//=============================================================================
// ST10_Flow4_B1Press.scl
// 1:1 CONVERSION FROM TIA PORTAL V18 GRAPH XML
// Generated: 2026-02-02
//=============================================================================

TYPE
    E_STEP_ST10_Flow4_B1Press : (
        STEP_ST10_Flow4_B1Press_F4_Initial := 1,
        STEP_ST10_Flow4_B1Press_ResultOKData := 145,
        STEP_ST10_Flow4_B1Press_MES_Check_NG := 306,
        STEP_ST10_Flow4_B1Press_Wait__robot_finish_task_1 := 134,
        STEP_ST10_Flow4_B1Press_B_PressFitting_01CylinderToHP_1 := 140,
        STEP_ST10_Flow4_B1Press_S2 := 2,
        STEP_ST10_Flow4_B1Press_Wait_robot_finish_task := 131,
        STEP_ST10_Flow4_B1Press_Step15 := 24,
        STEP_ST10_Flow4_B1Press_ShaftAndRingOK := 16,
        STEP_ST10_Flow4_B1Press_MesCheckIn := 304,
        STEP_ST10_Flow4_B1Press_MesCheckResult := 309,
        STEP_ST10_Flow4_B1Press_Step314 := 316,
        STEP_ST10_Flow4_B1Press_Status_Alarm := 118,
        STEP_ST10_Flow4_B1Press_StartCycle := 141,
        STEP_ST10_Flow4_B1Press_PressProgram := 8,
        STEP_ST10_Flow4_B1Press_Step400 := 400,
        STEP_ST10_Flow4_B1Press_NGCount := 404,
        STEP_ST10_Flow4_B1Press_RobotLeavePress_Area := 115,
        STEP_ST10_Flow4_B1Press_PartStatus_1 := 137,
        STEP_ST10_Flow4_B1Press_Part_Check := 239,
        STEP_ST10_Flow4_B1Press_MESOverTime := 315,
        STEP_ST10_Flow4_B1Press_B_PressFitting_01GripperCylinderToHP := 116,
        STEP_ST10_Flow4_B1Press_MES_Check_NG_1 := 310,
        STEP_ST10_Flow4_B1Press_MESOK := 19,
        STEP_ST10_Flow4_B1Press_Bypass_1 := 314,
        STEP_ST10_Flow4_B1Press_Request_robot_putShaft := 112,
        STEP_ST10_Flow4_B1Press_ok_1 := 317,
        STEP_ST10_Flow4_B1Press_CheckPressSensor := 138,
        STEP_ST10_Flow4_B1Press_PartCheck := 238,
        STEP_ST10_Flow4_B1Press_Pressing := 200,
        STEP_ST10_Flow4_B1Press_Request_robot_pick := 408,
        STEP_ST10_Flow4_B1Press_ProcessStart := 100,
        STEP_ST10_Flow4_B1Press_MES := 18,
        STEP_ST10_Flow4_B1Press_CheckPressGripStatus := 15,
        STEP_ST10_Flow4_B1Press_MES_1 := 25,
        STEP_ST10_Flow4_B1Press_ProcessFinish := 403,
        STEP_ST10_Flow4_B1Press_MESOverTime_1 := 312,
        STEP_ST10_Flow4_B1Press_DataMove := 132,
        STEP_ST10_Flow4_B1Press_Wait_robot_in_safety_area := 133,
        STEP_ST10_Flow4_B1Press_PutRing := 127,
        STEP_ST10_Flow4_B1Press_PressProgram_1 := 20,
        STEP_ST10_Flow4_B1Press_PressHoming := 9,
        STEP_ST10_Flow4_B1Press_MES__Check___In := 150,
        STEP_ST10_Flow4_B1Press_ShaftOK := 125,
        STEP_ST10_Flow4_B1Press_B_PressFitting_01CylinderToHP := 120,
        STEP_ST10_Flow4_B1Press_ProcessFInish_1 := 143,
        STEP_ST10_Flow4_B1Press_ResetMesCheckRequest := 301,
        STEP_ST10_Flow4_B1Press_CheckPressProgram := 139,
        STEP_ST10_Flow4_B1Press_CheckPressResult := 144,
        STEP_ST10_Flow4_B1Press_OKCount := 402,
        STEP_ST10_Flow4_B1Press_PressHoming_ := 13,
        STEP_ST10_Flow4_B1Press_MES_Result := 500,
        STEP_ST10_Flow4_B1Press_ProcessFinsh := 605,
        STEP_ST10_Flow4_B1Press_Request_robot_putRing := 113,
        STEP_ST10_Flow4_B1Press_StatusAlarm := 126,
        STEP_ST10_Flow4_B1Press_WaitPressFinish := 201,
        STEP_ST10_Flow4_B1Press_S3 := 3,
        STEP_ST10_Flow4_B1Press_Step147 := 147,
        STEP_ST10_Flow4_B1Press_PressReady__1 := 22,
        STEP_ST10_Flow4_B1Press_PressHoming_1 := 21,
        STEP_ST10_Flow4_B1Press_DataClear := 604,
        STEP_ST10_Flow4_B1Press_B_PressFitting_01GripperCylinderToWP := 119,
        STEP_ST10_Flow4_B1Press_Step313 := 313,
        STEP_ST10_Flow4_B1Press_ProductCheckAlarm := 240,
        STEP_ST10_Flow4_B1Press_CheckRingExist := 117,
        STEP_ST10_Flow4_B1Press_ProcessStart_CTStart := 104,
        STEP_ST10_Flow4_B1Press_RobotPick := 600,
        STEP_ST10_Flow4_B1Press_MES_Result_OK_1 := 399,
        STEP_ST10_Flow4_B1Press_CheckPressReady := 208,
        STEP_ST10_Flow4_B1Press_ProductCheckAlarm_1 := 241,
        STEP_ST10_Flow4_B1Press_Step14 := 14,
        STEP_ST10_Flow4_B1Press_Process_FInish := 149,
        STEP_ST10_Flow4_B1Press_Prepare_MES_CheckData_1 := 307,
        STEP_ST10_Flow4_B1Press_ResetMesUnloadRequest_1 := 302,
        STEP_ST10_Flow4_B1Press_JudgeStatus := 401,
        STEP_ST10_Flow4_B1Press_ResultNGData := 146,
        STEP_ST10_Flow4_B1Press_CheckFinish := 308,
        STEP_ST10_Flow4_B1Press_Normal_mode := 103,
        STEP_ST10_Flow4_B1Press_Bypass := 311,
        STEP_ST10_Flow4_B1Press_S5_MESInitial := 5,
        STEP_ST10_Flow4_B1Press_NoPart := 129,
        STEP_ST10_Flow4_B1Press_Wait__robot_finish_task := 130,
        STEP_ST10_Flow4_B1Press_PressReady_ := 12,
        STEP_ST10_Flow4_B1Press_MES_Check_Finish := 599,
        STEP_ST10_Flow4_B1Press_S4 := 4,
        STEP_ST10_Flow4_B1Press_CheckMachineStatus := 102,
        STEP_ST10_Flow4_B1Press_Determine_product_status := 101,
        STEP_ST10_Flow4_B1Press_Press_NG := 17,
        STEP_ST10_Flow4_B1Press_ResetPressStart := 142,
        STEP_ST10_Flow4_B1Press_PartStatus := 123,
        STEP_ST10_Flow4_B1Press_PressHoming__1 := 23,
        STEP_ST10_Flow4_B1Press_RobotLeavePressArea := 121,
        STEP_ST10_Flow4_B1Press_S10_InitialFinish := 10,
        STEP_ST10_Flow4_B1Press_Prepare_MES_CheckData := 303,
    ) INT := 1;
END_TYPE

CONST
    STEP_ST10_Flow4_B1Press_F4_Initial := 1;
    STEP_ST10_Flow4_B1Press_ResultOKData := 145;
    STEP_ST10_Flow4_B1Press_MES_Check_NG := 306;
    STEP_ST10_Flow4_B1Press_Wait__robot_finish_task_1 := 134;
    STEP_ST10_Flow4_B1Press_B_PressFitting_01CylinderToHP_1 := 140;
    STEP_ST10_Flow4_B1Press_S2 := 2;
    STEP_ST10_Flow4_B1Press_Wait_robot_finish_task := 131;
    STEP_ST10_Flow4_B1Press_Step15 := 24;
    STEP_ST10_Flow4_B1Press_ShaftAndRingOK := 16;
    STEP_ST10_Flow4_B1Press_MesCheckIn := 304;
    STEP_ST10_Flow4_B1Press_MesCheckResult := 309;
    STEP_ST10_Flow4_B1Press_Step314 := 316;
    STEP_ST10_Flow4_B1Press_Status_Alarm := 118;
    STEP_ST10_Flow4_B1Press_StartCycle := 141;
    STEP_ST10_Flow4_B1Press_PressProgram := 8;
    STEP_ST10_Flow4_B1Press_Step400 := 400;
    STEP_ST10_Flow4_B1Press_NGCount := 404;
    STEP_ST10_Flow4_B1Press_RobotLeavePress_Area := 115;
    STEP_ST10_Flow4_B1Press_PartStatus_1 := 137;
    STEP_ST10_Flow4_B1Press_Part_Check := 239;
    STEP_ST10_Flow4_B1Press_MESOverTime := 315;
    STEP_ST10_Flow4_B1Press_B_PressFitting_01GripperCylinderToHP := 116;
    STEP_ST10_Flow4_B1Press_MES_Check_NG_1 := 310;
    STEP_ST10_Flow4_B1Press_MESOK := 19;
    STEP_ST10_Flow4_B1Press_Bypass_1 := 314;
    STEP_ST10_Flow4_B1Press_Request_robot_putShaft := 112;
    STEP_ST10_Flow4_B1Press_ok_1 := 317;
    STEP_ST10_Flow4_B1Press_CheckPressSensor := 138;
    STEP_ST10_Flow4_B1Press_PartCheck := 238;
    STEP_ST10_Flow4_B1Press_Pressing := 200;
    STEP_ST10_Flow4_B1Press_Request_robot_pick := 408;
    STEP_ST10_Flow4_B1Press_ProcessStart := 100;
    STEP_ST10_Flow4_B1Press_MES := 18;
    STEP_ST10_Flow4_B1Press_CheckPressGripStatus := 15;
    STEP_ST10_Flow4_B1Press_MES_1 := 25;
    STEP_ST10_Flow4_B1Press_ProcessFinish := 403;
    STEP_ST10_Flow4_B1Press_MESOverTime_1 := 312;
    STEP_ST10_Flow4_B1Press_DataMove := 132;
    STEP_ST10_Flow4_B1Press_Wait_robot_in_safety_area := 133;
    STEP_ST10_Flow4_B1Press_PutRing := 127;
    STEP_ST10_Flow4_B1Press_PressProgram_1 := 20;
    STEP_ST10_Flow4_B1Press_PressHoming := 9;
    STEP_ST10_Flow4_B1Press_MES__Check___In := 150;
    STEP_ST10_Flow4_B1Press_ShaftOK := 125;
    STEP_ST10_Flow4_B1Press_B_PressFitting_01CylinderToHP := 120;
    STEP_ST10_Flow4_B1Press_ProcessFInish_1 := 143;
    STEP_ST10_Flow4_B1Press_ResetMesCheckRequest := 301;
    STEP_ST10_Flow4_B1Press_CheckPressProgram := 139;
    STEP_ST10_Flow4_B1Press_CheckPressResult := 144;
    STEP_ST10_Flow4_B1Press_OKCount := 402;
    STEP_ST10_Flow4_B1Press_PressHoming_ := 13;
    STEP_ST10_Flow4_B1Press_MES_Result := 500;
    STEP_ST10_Flow4_B1Press_ProcessFinsh := 605;
    STEP_ST10_Flow4_B1Press_Request_robot_putRing := 113;
    STEP_ST10_Flow4_B1Press_StatusAlarm := 126;
    STEP_ST10_Flow4_B1Press_WaitPressFinish := 201;
    STEP_ST10_Flow4_B1Press_S3 := 3;
    STEP_ST10_Flow4_B1Press_Step147 := 147;
    STEP_ST10_Flow4_B1Press_PressReady__1 := 22;
    STEP_ST10_Flow4_B1Press_PressHoming_1 := 21;
    STEP_ST10_Flow4_B1Press_DataClear := 604;
    STEP_ST10_Flow4_B1Press_B_PressFitting_01GripperCylinderToWP := 119;
    STEP_ST10_Flow4_B1Press_Step313 := 313;
    STEP_ST10_Flow4_B1Press_ProductCheckAlarm := 240;
    STEP_ST10_Flow4_B1Press_CheckRingExist := 117;
    STEP_ST10_Flow4_B1Press_ProcessStart_CTStart := 104;
    STEP_ST10_Flow4_B1Press_RobotPick := 600;
    STEP_ST10_Flow4_B1Press_MES_Result_OK_1 := 399;
    STEP_ST10_Flow4_B1Press_CheckPressReady := 208;
    STEP_ST10_Flow4_B1Press_ProductCheckAlarm_1 := 241;
    STEP_ST10_Flow4_B1Press_Step14 := 14;
    STEP_ST10_Flow4_B1Press_Process_FInish := 149;
    STEP_ST10_Flow4_B1Press_Prepare_MES_CheckData_1 := 307;
    STEP_ST10_Flow4_B1Press_ResetMesUnloadRequest_1 := 302;
    STEP_ST10_Flow4_B1Press_JudgeStatus := 401;
    STEP_ST10_Flow4_B1Press_ResultNGData := 146;
    STEP_ST10_Flow4_B1Press_CheckFinish := 308;
    STEP_ST10_Flow4_B1Press_Normal_mode := 103;
    STEP_ST10_Flow4_B1Press_Bypass := 311;
    STEP_ST10_Flow4_B1Press_S5_MESInitial := 5;
    STEP_ST10_Flow4_B1Press_NoPart := 129;
    STEP_ST10_Flow4_B1Press_Wait__robot_finish_task := 130;
    STEP_ST10_Flow4_B1Press_PressReady_ := 12;
    STEP_ST10_Flow4_B1Press_MES_Check_Finish := 599;
    STEP_ST10_Flow4_B1Press_S4 := 4;
    STEP_ST10_Flow4_B1Press_CheckMachineStatus := 102;
    STEP_ST10_Flow4_B1Press_Determine_product_status := 101;
    STEP_ST10_Flow4_B1Press_Press_NG := 17;
    STEP_ST10_Flow4_B1Press_ResetPressStart := 142;
    STEP_ST10_Flow4_B1Press_PartStatus := 123;
    STEP_ST10_Flow4_B1Press_PressHoming__1 := 23;
    STEP_ST10_Flow4_B1Press_RobotLeavePressArea := 121;
    STEP_ST10_Flow4_B1Press_S10_InitialFinish := 10;
    STEP_ST10_Flow4_B1Press_Prepare_MES_CheckData := 303;
END_CONST

FUNCTION_BLOCK "ST10_Flow4_B1Press_1to1"
{ S7_Optimized_Access := 'TRUE' }
VERSION : 1.0

VAR_INPUT
    iSysInface : "RCS_SysComInterface_V1";
END_VAR

VAR_IN_OUT
    ioPM_Inface : "RCS_PMInterface_V1";
    ioStatus : Int;
END_VAR

VAR_OUTPUT
    oAlarmID : Int;
END_VAR

VAR
    State : INT := 1;
    act_InitialRun : Bool;
    act_InitialOK : Bool;
    act_WaitRunning : Bool;
    act_Running : Bool;
    act_ProcessComplete : Bool;
    act_ProcessStart : Bool;
    act_UnPause : Bool;
    bError : Bool;
    wErrorID : Word;
END_VAR

BEGIN
    //======================================================================
    // STATE MACHINE - Inline Transition Conditions
    //======================================================================

    CASE #State OF

        // ===========================================
        // STEP 1: F4_Initial
        // ===========================================
        STEP_ST10_Flow4_B1Press_F4_Initial:
            // Action Qualifier=S
            // Token: #ioPM_Inface.InitialRun
            #ioPM_Inface.InitialRun := TRUE;
            // Action Qualifier=R
            // Token: #ioPM_Inface.InitialOK
            #ioPM_Inface.InitialOK := FALSE;
            // Action Qualifier=R
            // Token: #ioPM_Inface.WaitRunning
            #ioPM_Inface.WaitRunning := FALSE;
            // Action Qualifier=R
            // Token: #ioPM_Inface.Running
            #ioPM_Inface.Running := FALSE;
            // Action Qualifier=R
            // Token: #ioPM_Inface.UnPause
            #ioPM_Inface.UnPause := FALSE;
            // Action Qualifier=R
            // Token: "Station_Sys".Cmd.Calibration
            "Station_Sys".Cmd.Calibration := FALSE;
            // Action Qualifier=R
            // Token: "Station_Sys".Cmd.ChangeOver
            "Station_Sys".Cmd.ChangeOver := FALSE;
            // Action Qualifier=N
            // Token: //"ST350_Sys".Cmd.DryRun
            //"ST350_Sys".Cmd.DryRun;
            // Action Qualifier=R
            // Token: "Station_Sys".Cmd.Reserve
            "Station_Sys".Cmd.Reserve := FALSE;
            // Action Qualifier=R
            // Token: "Station_Sys".Cmd.OneCycle
            "Station_Sys".Cmd.OneCycle := FALSE;
            // Action Qualifier=R
            // Token: "DB_maXYmosNC1".StartCycle
            "DB_maXYmosNC1".StartCycle := FALSE;
            // Action Qualifier=R
            // Token: "DB_maXYmosNC1".StartCycle
            "DB_maXYmosNC1".StartCycle := FALSE;
            // Action Qualifier=R
            // Token: #ioPM_Inface.ProcessComplete
            #ioPM_Inface.ProcessComplete := FALSE;
            // Action Qualifier=R
            // Token: #ioPM_Inface.ProcessStart
            #ioPM_Inface.ProcessStart := FALSE;
            // Action Qualifier=R
            // Token: "AutoProcessControl".B_Press_1.Robot1PickPrimit
            "AutoProcessControl".B_Press_1.Robot1PickPrimit := FALSE;
            // Action Qualifier=R
            // Token: "AutoProcessControl".B_Press_1.Robot1PutShaftPrimit
            "AutoProcessControl".B_Press_1.Robot1PutShaftPrimit := FALSE;
            // Action Qualifier=R
            // Token: "AutoProcessControl".B_Press_1.Robot1PutRingPrimit
            "AutoProcessControl".B_Press_1.Robot1PutRingPrimit := FALSE;

            // Transition to next step: 145
            IF TRUE THEN  // Sequential transition - review XML for actual condition
                #State := STEP_ST10_Flow4_B1Press_ResultOKData;
            END_IF;

        // ===========================================
        // STEP 145: ResultOKData
        // ===========================================
        STEP_ST10_Flow4_B1Press_ResultOKData:
            // Action Qualifier=N
            // Token: "AutoProcessData".B_Press1.PartStatus := 280
            "AutoProcessData".B_Press1.PartStatus := 280;

            // Transition to next step: 306
            IF TRUE THEN  // Sequential transition - review XML for actual condition
                #State := STEP_ST10_Flow4_B1Press_MES_Check_NG;
            END_IF;

        // ===========================================
        // STEP 306: MES Check NG
        // ===========================================
        STEP_ST10_Flow4_B1Press_MES_Check_NG:
            // Action Qualifier=N
            // Token: "AutoProcessData".B_Press1.PartStatus := 251
            "AutoProcessData".B_Press1.PartStatus := 251;

            // Transition to next step: 134
            IF TRUE THEN  // Sequential transition - review XML for actual condition
                #State := STEP_ST10_Flow4_B1Press_Wait__robot_finish_task_1;
            END_IF;

        // ===========================================
        // STEP 134: Wait  robot finish task_1
        // ===========================================
        STEP_ST10_Flow4_B1Press_Wait__robot_finish_task_1:
            // No actions in XML

            // Transition to next step: 140
            IF TRUE THEN  // Sequential transition - review XML for actual condition
                #State := STEP_ST10_Flow4_B1Press_B_PressFitting_01CylinderToHP_1;
            END_IF;

        // ===========================================
        // STEP 140: B-PressFitting-01CylinderToHP_1
        // ===========================================
        STEP_ST10_Flow4_B1Press_B_PressFitting_01CylinderToHP_1:
            // Action Qualifier=S
            // Token: "ST10Cylinder".Cy[6].Inout.AutoGoHome
            "ST10Cylinder".Cy[6].Inout.AutoGoHome := TRUE;
            // Action Qualifier=R
            // Token: "ST10Cylinder".Cy[6].Inout.AutoGoWork
            "ST10Cylinder".Cy[6].Inout.AutoGoWork := FALSE;

            // Transition to next step: 2
            IF TRUE THEN  // Sequential transition - review XML for actual condition
                #State := STEP_ST10_Flow4_B1Press_S2;
            END_IF;

        // ===========================================
        // STEP 2: S2
        // ===========================================
        STEP_ST10_Flow4_B1Press_S2:
            // No actions in XML

            // Transition to next step: 131
            IF TRUE THEN  // Sequential transition - review XML for actual condition
                #State := STEP_ST10_Flow4_B1Press_Wait_robot_finish_task;
            END_IF;

        // ===========================================
        // STEP 131: Wait robot finish task
        // ===========================================
        STEP_ST10_Flow4_B1Press_Wait_robot_finish_task:
            // No actions in XML

            // Transition to next step: 24
            IF TRUE THEN  // Sequential transition - review XML for actual condition
                #State := STEP_ST10_Flow4_B1Press_Step15;
            END_IF;

        // ===========================================
        // STEP 24: Step15
        // ===========================================
        STEP_ST10_Flow4_B1Press_Step15:
            // No actions in XML

            // Transition to next step: 16
            IF TRUE THEN  // Sequential transition - review XML for actual condition
                #State := STEP_ST10_Flow4_B1Press_ShaftAndRingOK;
            END_IF;

        // ===========================================
        // STEP 16: ShaftAndRingOK
        // ===========================================
        STEP_ST10_Flow4_B1Press_ShaftAndRingOK:
            // No actions in XML

            // Transition to next step: 304
            IF TRUE THEN  // Sequential transition - review XML for actual condition
                #State := STEP_ST10_Flow4_B1Press_MesCheckIn;
            END_IF;

        // ===========================================
        // STEP 304: MesCheckIn
        // ===========================================
        STEP_ST10_Flow4_B1Press_MesCheckIn:
            // Action Qualifier=N
            // Token: "PLCtoMES"."PLC.Load_Station3ChickInReq"
            "PLCtoMES"."PLC.Load_Station3ChickInReq";

            // Transition to next step: 309
            IF TRUE THEN  // Sequential transition - review XML for actual condition
                #State := STEP_ST10_Flow4_B1Press_MesCheckResult;
            END_IF;

        // ===========================================
        // STEP 309: MesCheckResult
        // ===========================================
        STEP_ST10_Flow4_B1Press_MesCheckResult:
            // Action Qualifier=N
            // Token: "PLCtoMES"."PLC.Unload_Station3DataSaveReq"
            "PLCtoMES"."PLC.Unload_Station3DataSaveReq";

            // Transition to next step: 316
            IF TRUE THEN  // Sequential transition - review XML for actual condition
                #State := STEP_ST10_Flow4_B1Press_Step314;
            END_IF;

        // ===========================================
        // STEP 316: Step314
        // ===========================================
        STEP_ST10_Flow4_B1Press_Step314:
            // No actions in XML

            // Transition to next step: 118
            IF TRUE THEN  // Sequential transition - review XML for actual condition
                #State := STEP_ST10_Flow4_B1Press_Status_Alarm;
            END_IF;

        // ===========================================
        // STEP 118: Status Alarm
        // ===========================================
        STEP_ST10_Flow4_B1Press_Status_Alarm:
            // Action Qualifier=S
            // Token: "ST10_DeviceError".B.B1Press.StatusError
            "ST10_DeviceError".B.B1Press.StatusError := TRUE;

            // Transition to next step: 141
            IF TRUE THEN  // Sequential transition - review XML for actual condition
                #State := STEP_ST10_Flow4_B1Press_StartCycle;
            END_IF;

        // ===========================================
        // STEP 141: StartCycle
        // ===========================================
        STEP_ST10_Flow4_B1Press_StartCycle:
            // Action Qualifier=S
            // Token: "DB_maXYmosNC1".StartCycle
            "DB_maXYmosNC1".StartCycle := TRUE;

            // Transition to next step: 8
            IF TRUE THEN  // Sequential transition - review XML for actual condition
                #State := STEP_ST10_Flow4_B1Press_PressProgram;
            END_IF;

        // ===========================================
        // STEP 8: PressProgram
        // ===========================================
        STEP_ST10_Flow4_B1Press_PressProgram:
            // Action Qualifier=N
            // Token: "DB_maXYmosNC1".ProgNo := 1
            "DB_maXYmosNC1".ProgNo := 1;

            // Transition to next step: 400
            IF TRUE THEN  // Sequential transition - review XML for actual condition
                #State := STEP_ST10_Flow4_B1Press_Step400;
            END_IF;

        // ===========================================
        // STEP 400: Step400
        // ===========================================
        STEP_ST10_Flow4_B1Press_Step400:
            // No actions in XML

            // Transition to next step: 404
            IF TRUE THEN  // Sequential transition - review XML for actual condition
                #State := STEP_ST10_Flow4_B1Press_NGCount;
            END_IF;

        // ===========================================
        // STEP 404: NGCount
        // ===========================================
        STEP_ST10_Flow4_B1Press_NGCount:
            // Action Qualifier=N
            // Token: #ioPM_Inface.ProcessResult := #ioStatus
            #ioPM_Inface.ProcessResult := #ioStatus;

            // Transition to next step: 115
            IF TRUE THEN  // Sequential transition - review XML for actual condition
                #State := STEP_ST10_Flow4_B1Press_RobotLeavePress_Area;
            END_IF;

        // ===========================================
        // STEP 115: RobotLeavePress Area
        // ===========================================
        STEP_ST10_Flow4_B1Press_RobotLeavePress_Area:
            // No actions in XML

            // Transition to next step: 137
            IF TRUE THEN  // Sequential transition - review XML for actual condition
                #State := STEP_ST10_Flow4_B1Press_PartStatus_1;
            END_IF;

        // ===========================================
        // STEP 137: PartStatus_1
        // ===========================================
        STEP_ST10_Flow4_B1Press_PartStatus_1:
            // Action Qualifier=N
            // Token: "AutoProcessData".B_Press1.PartStatus := 250
            "AutoProcessData".B_Press1.PartStatus := 250;

            // Transition to next step: 239
            IF TRUE THEN  // Sequential transition - review XML for actual condition
                #State := STEP_ST10_Flow4_B1Press_Part_Check;
            END_IF;

        // ===========================================
        // STEP 239: Part Check
        // ===========================================
        STEP_ST10_Flow4_B1Press_Part_Check:
            // No actions in XML

            // Transition to next step: 315
            IF TRUE THEN  // Sequential transition - review XML for actual condition
                #State := STEP_ST10_Flow4_B1Press_MESOverTime;
            END_IF;

        // ===========================================
        // STEP 315: MESOverTime
        // ===========================================
        STEP_ST10_Flow4_B1Press_MESOverTime:
            // Action Qualifier=S
            // Token: "ST10_DeviceError".MES_Error.CheckInResultOverTime_3
            "ST10_DeviceError".MES_Error.CheckInResultOverTime_3 := TRUE;

            // Transition to next step: 116
            IF TRUE THEN  // Sequential transition - review XML for actual condition
                #State := STEP_ST10_Flow4_B1Press_B_PressFitting_01GripperCylinderToHP;
            END_IF;

        // ===========================================
        // STEP 116: B-PressFitting-01GripperCylinderToHP
        // ===========================================
        STEP_ST10_Flow4_B1Press_B_PressFitting_01GripperCylinderToHP:
            // Action Qualifier=S
            // Token: "ST10Cylinder".Cy[5].Inout.AutoGoHome
            "ST10Cylinder".Cy[5].Inout.AutoGoHome := TRUE;
            // Action Qualifier=R
            // Token: "ST10Cylinder".Cy[5].Inout.AutoGoWork
            "ST10Cylinder".Cy[5].Inout.AutoGoWork := FALSE;

            // Transition to next step: 310
            IF TRUE THEN  // Sequential transition - review XML for actual condition
                #State := STEP_ST10_Flow4_B1Press_MES_Check_NG_1;
            END_IF;

        // ===========================================
        // STEP 310: MES Check NG_1
        // ===========================================
        STEP_ST10_Flow4_B1Press_MES_Check_NG_1:
            // Action Qualifier=N
            // Token: "AutoProcessData".B_Press1.PartStatus := 252
            "AutoProcessData".B_Press1.PartStatus := 252;

            // Transition to next step: 19
            IF TRUE THEN  // Sequential transition - review XML for actual condition
                #State := STEP_ST10_Flow4_B1Press_MESOK;
            END_IF;

        // ===========================================
        // STEP 19: MESOK
        // ===========================================
        STEP_ST10_Flow4_B1Press_MESOK:
            // No actions in XML

            // Transition to next step: 314
            IF TRUE THEN  // Sequential transition - review XML for actual condition
                #State := STEP_ST10_Flow4_B1Press_Bypass_1;
            END_IF;

        // ===========================================
        // STEP 314: Bypass_1
        // ===========================================
        STEP_ST10_Flow4_B1Press_Bypass_1:
            // No actions in XML

            // Transition to next step: 112
            IF TRUE THEN  // Sequential transition - review XML for actual condition
                #State := STEP_ST10_Flow4_B1Press_Request_robot_putShaft;
            END_IF;

        // ===========================================
        // STEP 112: Request robot putShaft
        // ===========================================
        STEP_ST10_Flow4_B1Press_Request_robot_putShaft:
            // Action Qualifier=N
            // Token: "AutoProcessControl".B_Press_1.Robot1PutShaftPrimit
            "AutoProcessControl".B_Press_1.Robot1PutShaftPrimit;

            // Transition to next step: 317
            IF TRUE THEN  // Sequential transition - review XML for actual condition
                #State := STEP_ST10_Flow4_B1Press_ok_1;
            END_IF;

        // ===========================================
        // STEP 317: ok_1
        // ===========================================
        STEP_ST10_Flow4_B1Press_ok_1:
            // Action Qualifier=N
            // Token: "AutoProcessData".B_Press1.PartStatus := 299
            "AutoProcessData".B_Press1.PartStatus := 299;

            // Transition to next step: 138
            IF TRUE THEN  // Sequential transition - review XML for actual condition
                #State := STEP_ST10_Flow4_B1Press_CheckPressSensor;
            END_IF;

        // ===========================================
        // STEP 138: CheckPressSensor
        // ===========================================
        STEP_ST10_Flow4_B1Press_CheckPressSensor:
            // No actions in XML

            // Transition to next step: 238
            IF TRUE THEN  // Sequential transition - review XML for actual condition
                #State := STEP_ST10_Flow4_B1Press_PartCheck;
            END_IF;

        // ===========================================
        // STEP 238: PartCheck
        // ===========================================
        STEP_ST10_Flow4_B1Press_PartCheck:
            // No actions in XML

            // Transition to next step: 200
            IF TRUE THEN  // Sequential transition - review XML for actual condition
                #State := STEP_ST10_Flow4_B1Press_Pressing;
            END_IF;

        // ===========================================
        // STEP 200: Pressing
        // ===========================================
        STEP_ST10_Flow4_B1Press_Pressing:
            // No actions in XML

            // Transition to next step: 408
            IF TRUE THEN  // Sequential transition - review XML for actual condition
                #State := STEP_ST10_Flow4_B1Press_Request_robot_pick;
            END_IF;

        // ===========================================
        // STEP 408: Request robot pick
        // ===========================================
        STEP_ST10_Flow4_B1Press_Request_robot_pick:
            // Action Qualifier=N
            // Token: "AutoProcessControl".B_Press_1.Robot1PickPrimit
            "AutoProcessControl".B_Press_1.Robot1PickPrimit;

            // Transition to next step: 100
            IF TRUE THEN  // Sequential transition - review XML for actual condition
                #State := STEP_ST10_Flow4_B1Press_ProcessStart;
            END_IF;

        // ===========================================
        // STEP 100: ProcessStart
        // ===========================================
        STEP_ST10_Flow4_B1Press_ProcessStart:
            // Action Qualifier=R
            // Token: #ioPM_Inface.InitialRun
            #ioPM_Inface.InitialRun := FALSE;
            // Action Qualifier=R
            // Token: #ioPM_Inface.ProcessComplete
            #ioPM_Inface.ProcessComplete := FALSE;
            // Action Qualifier=R
            // Token: #ioPM_Inface.ProcessStart
            #ioPM_Inface.ProcessStart := FALSE;
            // Action Qualifier=S
            // Token: #ioPM_Inface.InitialOK
            #ioPM_Inface.InitialOK := TRUE;
            // Action Qualifier=S
            // Token: #ioPM_Inface.WaitRunning
            #ioPM_Inface.WaitRunning := TRUE;
            // Action Qualifier=N, Event="S1"
            // Token: #ioPM_Inface.ProcessResult := 0
            #ioPM_Inface.ProcessResult := 0;
            // Action Qualifier=R
            // Token: "ST10_GeneralData".FlowControl_Handshake[4].Start
            "ST10_GeneralData".FlowControl_Handshake[4].Start := FALSE;
            // Action Qualifier=R
            // Token: "ST10_GeneralData".FlowControl_Handshake[4].Done
            "ST10_GeneralData".FlowControl_Handshake[4].Done := FALSE;
            // Action Qualifier=N
            // Token: "MES_CHeck_DB".Station_3.CheckStep := 0
            "MES_CHeck_DB".Station_3.CheckStep := 0;
            // Action Qualifier=N
            // Token: "MES_CHeck_DB".Station_3.ResultStep := 0
            "MES_CHeck_DB".Station_3.ResultStep := 0;

            // Transition to next step: 18
            IF TRUE THEN  // Sequential transition - review XML for actual condition
                #State := STEP_ST10_Flow4_B1Press_MES;
            END_IF;

        // ===========================================
        // STEP 18: MES
        // ===========================================
        STEP_ST10_Flow4_B1Press_MES:
            // No actions in XML

            // Transition to next step: 15
            IF TRUE THEN  // Sequential transition - review XML for actual condition
                #State := STEP_ST10_Flow4_B1Press_CheckPressGripStatus;
            END_IF;

        // ===========================================
        // STEP 15: CheckPressGripStatus
        // ===========================================
        STEP_ST10_Flow4_B1Press_CheckPressGripStatus:
            // No actions in XML

            // Transition to next step: 25
            IF TRUE THEN  // Sequential transition - review XML for actual condition
                #State := STEP_ST10_Flow4_B1Press_MES_1;
            END_IF;

        // ===========================================
        // STEP 25: MES_1
        // ===========================================
        STEP_ST10_Flow4_B1Press_MES_1:
            // No actions in XML

            // Transition to next step: 403
            IF TRUE THEN  // Sequential transition - review XML for actual condition
                #State := STEP_ST10_Flow4_B1Press_ProcessFinish;
            END_IF;

        // ===========================================
        // STEP 403: ProcessFinish
        // ===========================================
        STEP_ST10_Flow4_B1Press_ProcessFinish:
            // No actions in XML

            // Transition to next step: 312
            IF TRUE THEN  // Sequential transition - review XML for actual condition
                #State := STEP_ST10_Flow4_B1Press_MESOverTime_1;
            END_IF;

        // ===========================================
        // STEP 312: MESOverTime_1
        // ===========================================
        STEP_ST10_Flow4_B1Press_MESOverTime_1:
            // Action Qualifier=S
            // Token: "ST10_DeviceError".MES_Error.CheckInCompOverTime_3
            "ST10_DeviceError".MES_Error.CheckInCompOverTime_3 := TRUE;

            // Transition to next step: 132
            IF TRUE THEN  // Sequential transition - review XML for actual condition
                #State := STEP_ST10_Flow4_B1Press_DataMove;
            END_IF;

        // ===========================================
        // STEP 132: DataMove
        // ===========================================
        STEP_ST10_Flow4_B1Press_DataMove:
            // No actions in XML

            // Transition to next step: 133
            IF TRUE THEN  // Sequential transition - review XML for actual condition
                #State := STEP_ST10_Flow4_B1Press_Wait_robot_in_safety_area;
            END_IF;

        // ===========================================
        // STEP 133: Wait robot in safety area
        // ===========================================
        STEP_ST10_Flow4_B1Press_Wait_robot_in_safety_area:
            // No actions in XML

            // Transition to next step: 127
            IF TRUE THEN  // Sequential transition - review XML for actual condition
                #State := STEP_ST10_Flow4_B1Press_PutRing;
            END_IF;

        // ===========================================
        // STEP 127: PutRing
        // ===========================================
        STEP_ST10_Flow4_B1Press_PutRing:
            // No actions in XML

            // Transition to next step: 20
            IF TRUE THEN  // Sequential transition - review XML for actual condition
                #State := STEP_ST10_Flow4_B1Press_PressProgram_1;
            END_IF;

        // ===========================================
        // STEP 20: PressProgram_1
        // ===========================================
        STEP_ST10_Flow4_B1Press_PressProgram_1:
            // Action Qualifier=N
            // Token: "DB_maXYmosNC1".ProgNo := 1
            "DB_maXYmosNC1".ProgNo := 1;

            // Transition to next step: 9
            IF TRUE THEN  // Sequential transition - review XML for actual condition
                #State := STEP_ST10_Flow4_B1Press_PressHoming;
            END_IF;

        // ===========================================
        // STEP 9: PressHoming
        // ===========================================
        STEP_ST10_Flow4_B1Press_PressHoming:
            // Action Qualifier=N
            // Token: "DB_maXYmosNC1".Homing
            "DB_maXYmosNC1".Homing;

            // Transition to next step: 150
            IF TRUE THEN  // Sequential transition - review XML for actual condition
                #State := STEP_ST10_Flow4_B1Press_MES__Check___In;
            END_IF;

        // ===========================================
        // STEP 150: MES  Check   In
        // ===========================================
        STEP_ST10_Flow4_B1Press_MES__Check___In:
            // No actions in XML

            // Transition to next step: 125
            IF TRUE THEN  // Sequential transition - review XML for actual condition
                #State := STEP_ST10_Flow4_B1Press_ShaftOK;
            END_IF;

        // ===========================================
        // STEP 125: ShaftOK
        // ===========================================
        STEP_ST10_Flow4_B1Press_ShaftOK:
            // No actions in XML

            // Transition to next step: 120
            IF TRUE THEN  // Sequential transition - review XML for actual condition
                #State := STEP_ST10_Flow4_B1Press_B_PressFitting_01CylinderToHP;
            END_IF;

        // ===========================================
        // STEP 120: B-PressFitting-01CylinderToHP
        // ===========================================
        STEP_ST10_Flow4_B1Press_B_PressFitting_01CylinderToHP:
            // Action Qualifier=S
            // Token: "ST10Cylinder".Cy[6].Inout.AutoGoHome
            "ST10Cylinder".Cy[6].Inout.AutoGoHome := TRUE;
            // Action Qualifier=R
            // Token: "ST10Cylinder".Cy[6].Inout.AutoGoWork
            "ST10Cylinder".Cy[6].Inout.AutoGoWork := FALSE;

            // Transition to next step: 143
            IF TRUE THEN  // Sequential transition - review XML for actual condition
                #State := STEP_ST10_Flow4_B1Press_ProcessFInish_1;
            END_IF;

        // ===========================================
        // STEP 143: ProcessFInish 1
        // ===========================================
        STEP_ST10_Flow4_B1Press_ProcessFInish_1:
            // No actions in XML

            // Transition to next step: 301
            IF TRUE THEN  // Sequential transition - review XML for actual condition
                #State := STEP_ST10_Flow4_B1Press_ResetMesCheckRequest;
            END_IF;

        // ===========================================
        // STEP 301: ResetMesCheckRequest
        // ===========================================
        STEP_ST10_Flow4_B1Press_ResetMesCheckRequest:
            // Action Qualifier=R
            // Token: "PLCtoMES"."PLC.Load_Station3ChickInReq"
            "PLCtoMES"."PLC.Load_Station3ChickInReq" := FALSE;
            // Action Qualifier=R
            // Token: "MEStoPLC"."MES.Load_Station3PartOK"
            "MEStoPLC"."MES.Load_Station3PartOK" := FALSE;
            // Action Qualifier=R
            // Token: "MEStoPLC"."MES.Load_Station3PartNG"
            "MEStoPLC"."MES.Load_Station3PartNG" := FALSE;
            // Action Qualifier=R
            // Token: "MEStoPLC"."MES.Load_Station3ReqMesDone"
            "MEStoPLC"."MES.Load_Station3ReqMesDone" := FALSE;

            // Transition to next step: 139
            IF TRUE THEN  // Sequential transition - review XML for actual condition
                #State := STEP_ST10_Flow4_B1Press_CheckPressProgram;
            END_IF;

        // ===========================================
        // STEP 139: CheckPressProgram
        // ===========================================
        STEP_ST10_Flow4_B1Press_CheckPressProgram:
            // Action Qualifier=N
            // Token: "AutoProcessData".B_Press1.Press1Program := "DB_maXYmosNC1".InputMessages.StatusBits.MP
            "AutoProcessData".B_Press1.Press1Program := "DB_maXYmosNC1".InputMessages.StatusBits.MP;

            // Transition to next step: 144
            IF TRUE THEN  // Sequential transition - review XML for actual condition
                #State := STEP_ST10_Flow4_B1Press_CheckPressResult;
            END_IF;

        // ===========================================
        // STEP 144: CheckPressResult
        // ===========================================
        STEP_ST10_Flow4_B1Press_CheckPressResult:
            // No actions in XML

            // Transition to next step: 402
            IF TRUE THEN  // Sequential transition - review XML for actual condition
                #State := STEP_ST10_Flow4_B1Press_OKCount;
            END_IF;

        // ===========================================
        // STEP 402: OKCount
        // ===========================================
        STEP_ST10_Flow4_B1Press_OKCount:
            // Action Qualifier=N
            // Token: #ioPM_Inface.ProcessResult := 400
            #ioPM_Inface.ProcessResult := 400;

            // Transition to next step: 13
            IF TRUE THEN  // Sequential transition - review XML for actual condition
                #State := STEP_ST10_Flow4_B1Press_PressHoming_;
            END_IF;

        // ===========================================
        // STEP 13: PressHoming?
        // ===========================================
        STEP_ST10_Flow4_B1Press_PressHoming_:
            // No actions in XML

            // Transition to next step: 500
            IF TRUE THEN  // Sequential transition - review XML for actual condition
                #State := STEP_ST10_Flow4_B1Press_MES_Result;
            END_IF;

        // ===========================================
        // STEP 500: MES Result
        // ===========================================
        STEP_ST10_Flow4_B1Press_MES_Result:
            // No actions in XML

            // Transition to next step: 605
            IF TRUE THEN  // Sequential transition - review XML for actual condition
                #State := STEP_ST10_Flow4_B1Press_ProcessFinsh;
            END_IF;

        // ===========================================
        // STEP 605: ProcessFinsh
        // ===========================================
        STEP_ST10_Flow4_B1Press_ProcessFinsh:
            // No actions in XML

            // Transition to next step: 113
            IF TRUE THEN  // Sequential transition - review XML for actual condition
                #State := STEP_ST10_Flow4_B1Press_Request_robot_putRing;
            END_IF;

        // ===========================================
        // STEP 113: Request robot putRing
        // ===========================================
        STEP_ST10_Flow4_B1Press_Request_robot_putRing:
            // Action Qualifier=N
            // Token: "AutoProcessControl".B_Press_1.Robot1PutRingPrimit
            "AutoProcessControl".B_Press_1.Robot1PutRingPrimit;

            // Transition to next step: 126
            IF TRUE THEN  // Sequential transition - review XML for actual condition
                #State := STEP_ST10_Flow4_B1Press_StatusAlarm;
            END_IF;

        // ===========================================
        // STEP 126: StatusAlarm
        // ===========================================
        STEP_ST10_Flow4_B1Press_StatusAlarm:
            // Action Qualifier=S
            // Token: "ST10_DeviceError".B.B1Press.StatusError
            "ST10_DeviceError".B.B1Press.StatusError := TRUE;

            // Transition to next step: 201
            IF TRUE THEN  // Sequential transition - review XML for actual condition
                #State := STEP_ST10_Flow4_B1Press_WaitPressFinish;
            END_IF;

        // ===========================================
        // STEP 201: WaitPressFinish
        // ===========================================
        STEP_ST10_Flow4_B1Press_WaitPressFinish:
            // No actions in XML

            // Transition to next step: 3
            IF TRUE THEN  // Sequential transition - review XML for actual condition
                #State := STEP_ST10_Flow4_B1Press_S3;
            END_IF;

        // ===========================================
        // STEP 3: S3
        // ===========================================
        STEP_ST10_Flow4_B1Press_S3:
            // No actions in XML

            // Transition to next step: 147
            IF TRUE THEN  // Sequential transition - review XML for actual condition
                #State := STEP_ST10_Flow4_B1Press_Step147;
            END_IF;

        // ===========================================
        // STEP 147: Step147
        // ===========================================
        STEP_ST10_Flow4_B1Press_Step147:
            // No actions in XML

            // Transition to next step: 22
            IF TRUE THEN  // Sequential transition - review XML for actual condition
                #State := STEP_ST10_Flow4_B1Press_PressReady__1;
            END_IF;

        // ===========================================
        // STEP 22: PressReady?_1
        // ===========================================
        STEP_ST10_Flow4_B1Press_PressReady__1:
            // No actions in XML

            // Transition to next step: 21
            IF TRUE THEN  // Sequential transition - review XML for actual condition
                #State := STEP_ST10_Flow4_B1Press_PressHoming_1;
            END_IF;

        // ===========================================
        // STEP 21: PressHoming_1
        // ===========================================
        STEP_ST10_Flow4_B1Press_PressHoming_1:
            // Action Qualifier=N
            // Token: "DB_maXYmosNC1".Homing
            "DB_maXYmosNC1".Homing;

            // Transition to next step: 604
            IF TRUE THEN  // Sequential transition - review XML for actual condition
                #State := STEP_ST10_Flow4_B1Press_DataClear;
            END_IF;

        // ===========================================
        // STEP 604: DataClear
        // ===========================================
        STEP_ST10_Flow4_B1Press_DataClear:
            // Action Qualifier=N, Event="S1"
            // Token: #ioPM_Inface.ProcessResult := 0
            #ioPM_Inface.ProcessResult := 0;
            // Action Qualifier=N, Event="S1"
            // Token: #ioStatus := 0
            #ioStatus := 0;

            // Transition to next step: 119
            IF TRUE THEN  // Sequential transition - review XML for actual condition
                #State := STEP_ST10_Flow4_B1Press_B_PressFitting_01GripperCylinderToWP;
            END_IF;

        // ===========================================
        // STEP 119: B-PressFitting-01GripperCylinderToWP
        // ===========================================
        STEP_ST10_Flow4_B1Press_B_PressFitting_01GripperCylinderToWP:
            // Action Qualifier=R
            // Token: "ST10Cylinder".Cy[5].Inout.AutoGoHome
            "ST10Cylinder".Cy[5].Inout.AutoGoHome := FALSE;
            // Action Qualifier=S
            // Token: "ST10Cylinder".Cy[5].Inout.AutoGoWork
            "ST10Cylinder".Cy[5].Inout.AutoGoWork := TRUE;

            // Transition to next step: 313
            IF TRUE THEN  // Sequential transition - review XML for actual condition
                #State := STEP_ST10_Flow4_B1Press_Step313;
            END_IF;

        // ===========================================
        // STEP 313: Step313
        // ===========================================
        STEP_ST10_Flow4_B1Press_Step313:
            // No actions in XML

            // Transition to next step: 240
            IF TRUE THEN  // Sequential transition - review XML for actual condition
                #State := STEP_ST10_Flow4_B1Press_ProductCheckAlarm;
            END_IF;

        // ===========================================
        // STEP 240: ProductCheckAlarm
        // ===========================================
        STEP_ST10_Flow4_B1Press_ProductCheckAlarm:
            // Action Qualifier=S
            // Token: "ST10_DeviceError".B.B1Press.ShaftSensorCheckError
            "ST10_DeviceError".B.B1Press.ShaftSensorCheckError := TRUE;

            // Transition to next step: 117
            IF TRUE THEN  // Sequential transition - review XML for actual condition
                #State := STEP_ST10_Flow4_B1Press_CheckRingExist;
            END_IF;

        // ===========================================
        // STEP 117: CheckRingExist
        // ===========================================
        STEP_ST10_Flow4_B1Press_CheckRingExist:
            // No actions in XML

            // Transition to next step: 104
            IF TRUE THEN  // Sequential transition - review XML for actual condition
                #State := STEP_ST10_Flow4_B1Press_ProcessStart_CTStart;
            END_IF;

        // ===========================================
        // STEP 104: ProcessStart,CTStart
        // ===========================================
        STEP_ST10_Flow4_B1Press_ProcessStart_CTStart:
            // Action Qualifier=S
            // Token: #ioPM_Inface.ProcessStart
            #ioPM_Inface.ProcessStart := TRUE;
            // Action Qualifier=R
            // Token: #ioPM_Inface.ProcessComplete
            #ioPM_Inface.ProcessComplete := FALSE;

            // Transition to next step: 600
            IF TRUE THEN  // Sequential transition - review XML for actual condition
                #State := STEP_ST10_Flow4_B1Press_RobotPick;
            END_IF;

        // ===========================================
        // STEP 600: RobotPick
        // ===========================================
        STEP_ST10_Flow4_B1Press_RobotPick:
            // Action Qualifier=S
            // Token: #ioPM_Inface.ProcessComplete
            #ioPM_Inface.ProcessComplete := TRUE;
            // Action Qualifier=R
            // Token: #ioPM_Inface.ProcessStart
            #ioPM_Inface.ProcessStart := FALSE;

            // Transition to next step: 399
            IF TRUE THEN  // Sequential transition - review XML for actual condition
                #State := STEP_ST10_Flow4_B1Press_MES_Result_OK_1;
            END_IF;

        // ===========================================
        // STEP 399: MES Result OK_1
        // ===========================================
        STEP_ST10_Flow4_B1Press_MES_Result_OK_1:
            // Action Qualifier=N
            // Token: "AutoProcessData".B_Press1.PartStatus := 299
            "AutoProcessData".B_Press1.PartStatus := 299;

            // Transition to next step: 208
            IF TRUE THEN  // Sequential transition - review XML for actual condition
                #State := STEP_ST10_Flow4_B1Press_CheckPressReady;
            END_IF;

        // ===========================================
        // STEP 208: CheckPressReady
        // ===========================================
        STEP_ST10_Flow4_B1Press_CheckPressReady:
            // Action Qualifier=R
            // Token: "DB_maXYmosNC1".StartCycle
            "DB_maXYmosNC1".StartCycle := FALSE;

            // Transition to next step: 241
            IF TRUE THEN  // Sequential transition - review XML for actual condition
                #State := STEP_ST10_Flow4_B1Press_ProductCheckAlarm_1;
            END_IF;

        // ===========================================
        // STEP 241: ProductCheckAlarm_1
        // ===========================================
        STEP_ST10_Flow4_B1Press_ProductCheckAlarm_1:
            // Action Qualifier=S
            // Token: "ST10_DeviceError".B.B1Press.RingSensorCheckError
            "ST10_DeviceError".B.B1Press.RingSensorCheckError := TRUE;

            // Transition to next step: 14
            IF TRUE THEN  // Sequential transition - review XML for actual condition
                #State := STEP_ST10_Flow4_B1Press_Step14;
            END_IF;

        // ===========================================
        // STEP 14: Step14
        // ===========================================
        STEP_ST10_Flow4_B1Press_Step14:
            // No actions in XML

            // Transition to next step: 149
            IF TRUE THEN  // Sequential transition - review XML for actual condition
                #State := STEP_ST10_Flow4_B1Press_Process_FInish;
            END_IF;

        // ===========================================
        // STEP 149: Process FInish
        // ===========================================
        STEP_ST10_Flow4_B1Press_Process_FInish:
            // No actions in XML

            // Transition to next step: 307
            IF TRUE THEN  // Sequential transition - review XML for actual condition
                #State := STEP_ST10_Flow4_B1Press_Prepare_MES_CheckData_1;
            END_IF;

        // ===========================================
        // STEP 307: Prepare MES CheckData_1
        // ===========================================
        STEP_ST10_Flow4_B1Press_Prepare_MES_CheckData_1:
            // No actions in XML

            // Transition to next step: 302
            IF TRUE THEN  // Sequential transition - review XML for actual condition
                #State := STEP_ST10_Flow4_B1Press_ResetMesUnloadRequest_1;
            END_IF;

        // ===========================================
        // STEP 302: ResetMesUnloadRequest_1
        // ===========================================
        STEP_ST10_Flow4_B1Press_ResetMesUnloadRequest_1:
            // Action Qualifier=R
            // Token: "PLCtoMES"."PLC.Unload_Station3DataSaveReq"
            "PLCtoMES"."PLC.Unload_Station3DataSaveReq" := FALSE;
            // Action Qualifier=R
            // Token: "MEStoPLC"."MES.Unload_ResultsStored3OK"
            "MEStoPLC"."MES.Unload_ResultsStored3OK" := FALSE;
            // Action Qualifier=R
            // Token: "MEStoPLC"."MES.Unload_ResultsStored3NG"
            "MEStoPLC"."MES.Unload_ResultsStored3NG" := FALSE;
            // Action Qualifier=R
            // Token: "MEStoPLC"."MES.Unload_ResultsStored3ReqMesDone"
            "MEStoPLC"."MES.Unload_ResultsStored3ReqMesDone" := FALSE;

            // Transition to next step: 401
            IF TRUE THEN  // Sequential transition - review XML for actual condition
                #State := STEP_ST10_Flow4_B1Press_JudgeStatus;
            END_IF;

        // ===========================================
        // STEP 401: JudgeStatus
        // ===========================================
        STEP_ST10_Flow4_B1Press_JudgeStatus:
            // Action Qualifier=N
            // Token: #ioPM_Inface.ProcessResult := 0
            #ioPM_Inface.ProcessResult := 0;

            // Transition to next step: 146
            IF TRUE THEN  // Sequential transition - review XML for actual condition
                #State := STEP_ST10_Flow4_B1Press_ResultNGData;
            END_IF;

        // ===========================================
        // STEP 146: ResultNGData
        // ===========================================
        STEP_ST10_Flow4_B1Press_ResultNGData:
            // Action Qualifier=N
            // Token: "AutoProcessData".B_Press1.PartStatus := 255
            "AutoProcessData".B_Press1.PartStatus := 255;

            // Transition to next step: 308
            IF TRUE THEN  // Sequential transition - review XML for actual condition
                #State := STEP_ST10_Flow4_B1Press_CheckFinish;
            END_IF;

        // ===========================================
        // STEP 308: CheckFinish
        // ===========================================
        STEP_ST10_Flow4_B1Press_CheckFinish:
            // No actions in XML

            // Transition to next step: 103
            IF TRUE THEN  // Sequential transition - review XML for actual condition
                #State := STEP_ST10_Flow4_B1Press_Normal_mode;
            END_IF;

        // ===========================================
        // STEP 103: Normal mode
        // ===========================================
        STEP_ST10_Flow4_B1Press_Normal_mode:
            // No actions in XML

            // Transition to next step: 311
            IF TRUE THEN  // Sequential transition - review XML for actual condition
                #State := STEP_ST10_Flow4_B1Press_Bypass;
            END_IF;

        // ===========================================
        // STEP 311: Bypass
        // ===========================================
        STEP_ST10_Flow4_B1Press_Bypass:
            // No actions in XML

            // Transition to next step: 5
            IF TRUE THEN  // Sequential transition - review XML for actual condition
                #State := STEP_ST10_Flow4_B1Press_S5_MESInitial;
            END_IF;

        // ===========================================
        // STEP 5: S5_MESInitial
        // ===========================================
        STEP_ST10_Flow4_B1Press_S5_MESInitial:
            // No actions in XML

            // Transition to next step: 129
            IF TRUE THEN  // Sequential transition - review XML for actual condition
                #State := STEP_ST10_Flow4_B1Press_NoPart;
            END_IF;

        // ===========================================
        // STEP 129: NoPart
        // ===========================================
        STEP_ST10_Flow4_B1Press_NoPart:
            // No actions in XML

            // Transition to next step: 130
            IF TRUE THEN  // Sequential transition - review XML for actual condition
                #State := STEP_ST10_Flow4_B1Press_Wait__robot_finish_task;
            END_IF;

        // ===========================================
        // STEP 130: Wait  robot finish task
        // ===========================================
        STEP_ST10_Flow4_B1Press_Wait__robot_finish_task:
            // No actions in XML

            // Transition to next step: 12
            IF TRUE THEN  // Sequential transition - review XML for actual condition
                #State := STEP_ST10_Flow4_B1Press_PressReady_;
            END_IF;

        // ===========================================
        // STEP 12: PressReady?
        // ===========================================
        STEP_ST10_Flow4_B1Press_PressReady_:
            // No actions in XML

            // Transition to next step: 599
            IF TRUE THEN  // Sequential transition - review XML for actual condition
                #State := STEP_ST10_Flow4_B1Press_MES_Check_Finish;
            END_IF;

        // ===========================================
        // STEP 599: MES Check Finish
        // ===========================================
        STEP_ST10_Flow4_B1Press_MES_Check_Finish:
            // No actions in XML

            // Transition to next step: 4
            IF TRUE THEN  // Sequential transition - review XML for actual condition
                #State := STEP_ST10_Flow4_B1Press_S4;
            END_IF;

        // ===========================================
        // STEP 4: S4
        // ===========================================
        STEP_ST10_Flow4_B1Press_S4:
            // No actions in XML

            // Transition to next step: 102
            IF TRUE THEN  // Sequential transition - review XML for actual condition
                #State := STEP_ST10_Flow4_B1Press_CheckMachineStatus;
            END_IF;

        // ===========================================
        // STEP 102: CheckMachineStatus
        // ===========================================
        STEP_ST10_Flow4_B1Press_CheckMachineStatus:
            // No actions in XML

            // Transition to next step: 101
            IF TRUE THEN  // Sequential transition - review XML for actual condition
                #State := STEP_ST10_Flow4_B1Press_Determine_product_status;
            END_IF;

        // ===========================================
        // STEP 101: Determine product status
        // ===========================================
        STEP_ST10_Flow4_B1Press_Determine_product_status:
            // No actions in XML

            // Transition to next step: 17
            IF TRUE THEN  // Sequential transition - review XML for actual condition
                #State := STEP_ST10_Flow4_B1Press_Press_NG;
            END_IF;

        // ===========================================
        // STEP 17: Press NG
        // ===========================================
        STEP_ST10_Flow4_B1Press_Press_NG:
            // No actions in XML

            // Transition to next step: 142
            IF TRUE THEN  // Sequential transition - review XML for actual condition
                #State := STEP_ST10_Flow4_B1Press_ResetPressStart;
            END_IF;

        // ===========================================
        // STEP 142: ResetPressStart
        // ===========================================
        STEP_ST10_Flow4_B1Press_ResetPressStart:
            // Action Qualifier=R
            // Token: "DB_maXYmosNC1".StartCycle
            "DB_maXYmosNC1".StartCycle := FALSE;

            // Transition to next step: 123
            IF TRUE THEN  // Sequential transition - review XML for actual condition
                #State := STEP_ST10_Flow4_B1Press_PartStatus;
            END_IF;

        // ===========================================
        // STEP 123: PartStatus
        // ===========================================
        STEP_ST10_Flow4_B1Press_PartStatus:
            // No actions in XML

            // Transition to next step: 23
            IF TRUE THEN  // Sequential transition - review XML for actual condition
                #State := STEP_ST10_Flow4_B1Press_PressHoming__1;
            END_IF;

        // ===========================================
        // STEP 23: PressHoming?_1
        // ===========================================
        STEP_ST10_Flow4_B1Press_PressHoming__1:
            // No actions in XML

            // Transition to next step: 121
            IF TRUE THEN  // Sequential transition - review XML for actual condition
                #State := STEP_ST10_Flow4_B1Press_RobotLeavePressArea;
            END_IF;

        // ===========================================
        // STEP 121: RobotLeavePressArea
        // ===========================================
        STEP_ST10_Flow4_B1Press_RobotLeavePressArea:
            // No actions in XML

            // Transition to next step: 10
            IF TRUE THEN  // Sequential transition - review XML for actual condition
                #State := STEP_ST10_Flow4_B1Press_S10_InitialFinish;
            END_IF;

        // ===========================================
        // STEP 10: S10_InitialFinish
        // ===========================================
        STEP_ST10_Flow4_B1Press_S10_InitialFinish:
            // Action Qualifier=S
            // Token: #ioPM_Inface.InitialOK
            #ioPM_Inface.InitialOK := TRUE;

            // Transition to next step: 303
            IF TRUE THEN  // Sequential transition - review XML for actual condition
                #State := STEP_ST10_Flow4_B1Press_Prepare_MES_CheckData;
            END_IF;

        // ===========================================
        // STEP 303: Prepare MES CheckData
        // ===========================================
        STEP_ST10_Flow4_B1Press_Prepare_MES_CheckData:
            // No actions in XML

    END_CASE;

    // UPDATE ioPM_Inface
    #ioPM_Inface.InitialRun := #act_InitialRun;
    #ioPM_Inface.InitialOK := #act_InitialOK;
    #ioPM_Inface.WaitRunning := #act_WaitRunning;
    #ioPM_Inface.Running := #act_Running;
    #ioPM_Inface.ProcessComplete := #act_ProcessComplete;
    #ioPM_Inface.ProcessStart := #act_ProcessStart;
    #ioPM_Inface.UnPause := #act_UnPause;

    // ERROR HANDLING
    IF #bError THEN
        #ioStatus := 900;
        #oAlarmID := INT_TO_WORD(#wErrorID);
    ELSE
        #ioStatus := 0;
        #oAlarmID := 0;
    END_IF;
END_FUNCTION_BLOCK

//=============================================================================
// END OF FILE
//=============================================================================
